FUNCTION_BLOCK FB107
TITLE = ''
AUTHOR : CB

VAR
	modes : FB41;
	fault : FB68;
	process : FB79;
	pilot : FB106;
END_VAR


BEGIN


NETWORK
TITLE =
//
//	modes
CALL #modes;



NETWORK
TITLE =
//
//	fault
CALL #fault;



NETWORK
TITLE =
//
//	process
CALL #process;



NETWORK
TITLE =
//
//	pilot
CALL #pilot;




END_FUNCTION_BLOCK
